{attribute 'GeneratedUsingTerminal: IODEVICETYPE_ETHERCATPROT'}
{attribute addProperty BoxType "IODEVICETYPE_ETHERCATPROT"}
{attribute addProperty Id "Beckhoff_ELXxxxxBeckhoff_ELXxxxx_11EBC10B663SyncUnitsSyncUnits_99E584AF18InputsInputs_25A0042B160OutputsOutputs_2397A10E106InfoDataInfoData_C76BEFB322"}
{attribute addProperty CRC "3189232939"}
{attribute addProperty Size "969"}
TYPE EtherCAT_Master_ELXxxxx_BE17D52B :
STRUCT
	{attribute addProperty Name "Beckhoff_ELXxxxx"}
	{attribute addProperty PreviousPort "EtherCAT_Master_ELXxxxx : Master"}
	Beckhoff_ELXxxxx : Beckhoff_ELXxxxx_11EBC10B;
	{attribute addProperty Name "SyncUnits"}
	SyncUnits : SyncUnits_99E584AF;
	{attribute addProperty Name "Inputs"}
	Inputs : Inputs_25A0042B;
	{attribute addProperty Name "Outputs"}
	Outputs : Outputs_2397A10E;
	{attribute addProperty Name "InfoData"}
	InfoData : InfoData_C76BEFB3;
END_STRUCT
END_TYPE

(* stored: Version 1.2.0.0, ProductVersion 3.1.4024.9
   DUT EtherCAT_Master_ELXxxxx_BE17D52B: Id {c1d8de19-f58e-4f43-910c-e74fdbe9fc9c} *)
